{attribute 'qualified_only'}
VAR_GLOBAL
    
END_VAR

(* stored: Version 1.1.0.1, ProductVersion 3.1.4022.18
   GVL GVL_States: Id {0d66e36e-6edb-44aa-84ac-61e21899dbaf} *)
